FUNCTION_BLOCK Resize (* openCV resize *)
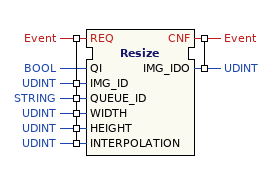
  EVENT_INPUT
    REQ WITH IMG_ID, QUEUE_ID, WIDTH, HEIGHT, INTERPOLATION;
  END_EVENT
  EVENT_OUTPUT
    CNF WITH IMG_IDO;
  END_EVENT
  VAR_INPUT
    QI : BOOL;
    IMG_ID : UDINT;
    QUEUE_ID : STRING;
    WIDTH : UDINT;
    HEIGHT : UDINT;
    INTERPOLATION : UDINT;
  END_VAR
  VAR_OUTPUT
    IMG_IDO : UDINT;
  END_VAR
END_FUNCTION_BLOCK
